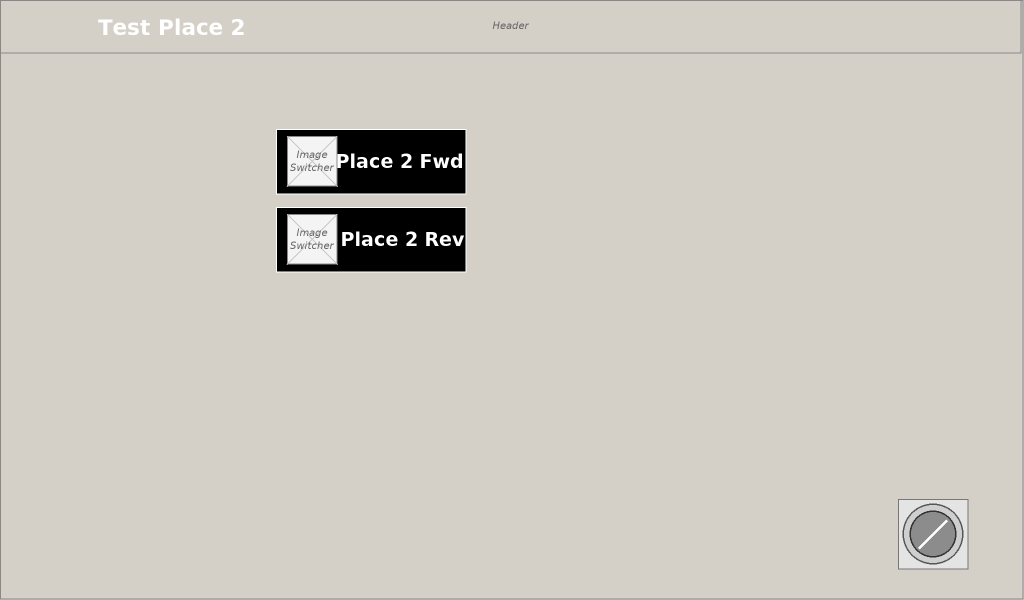
VISUALIZATION Test_Place2  // 1024x600
    Frame (0,-2 1021x55)
        shows Header()
    Label (95,15 250x25), "Test Place 2"
    RotarySwitch (898,499 70x70), variable: HMI_GVL.bTestModeEnablePlacing2, behaviour: TOGGLE, style: Switch-RotarySwitch-Gray
    RoundedRectangle (276,129 190x65)
        toggle Status_GVL.stMotor_Placing2.iTestForward
    Label (331,149 137x25), "Place 2 Fwd"
    ImageSwitcher (287,136 50x50), variable: Status_GVL.stMotor_Placing2.iTestForward, behaviour: TOGGLE
    RoundedRectangle (276,207 190x65)
        toggle Status_GVL.stMotor_Placing2.iTestReverse
    Label (334,227 137x25), "Place 2 Rev"
    ImageSwitcher (287,214 50x50), variable: Status_GVL.stMotor_Placing2.iTestReverse, behaviour: TOGGLE
END_VISUALIZATION

(* stored: Version 1.1.0.1, ProductVersion 3.1.4024.12
   Visu Test_Place2: Id {b75d3cfd-36a1-4cf1-8793-d996925cfb63} *)
